FUNCTION ASSEMBLE_BYTE_FROM_QUARTERS (* this Function combines the 4 QUARTER BYTES to a BYTE *)
  (* Standard: 61499-1; Description: Copyright (c) 2024 HR Agrartechnik GmbH This program and the accompanying materials are made available under the terms of the Eclipse Public License 2.0 which is available at https://www.eclipse.org/legal/epl-2.0/ SPDX-License-Identifier: EPL-2.0 *)
  (* Version 3.0, 2025-04-14, Patrick Aigner, changed package *)
  (* Version 1.1, 2024-07-28, Moritz Ortmeier, HR Agrartechnik, rename Function and change Input/Output Variables *)
  (* Version 1.0, 2024-02-22, Franz H??pfinger, HR Agrartechnik, initial Implementation *)
  PACKAGE eclipse4diac::utils::assembling;
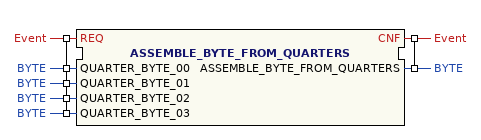
  EVENT_INPUT
    REQ WITH QUARTER_BYTE_00, QUARTER_BYTE_01, QUARTER_BYTE_02, QUARTER_BYTE_03;
  END_EVENT
  EVENT_OUTPUT
    CNF WITH ASSEMBLE_BYTE_FROM_QUARTERS;
  END_EVENT
  VAR_INPUT
    QUARTER_BYTE_00 : BYTE;
    QUARTER_BYTE_01 : BYTE;
    QUARTER_BYTE_02 : BYTE;
    QUARTER_BYTE_03 : BYTE;
  END_VAR
  VAR_OUTPUT
    ASSEMBLE_BYTE_FROM_QUARTERS : BYTE;
  END_VAR
  BODY IN ST:
(* this Function combines the 4 QUARTER BYTES to a BYTE *)
FUNCTION ASSEMBLE_BYTE_FROM_QUARTERS : BYTE

VAR_INPUT
	QUARTER_BYTE_00 : BYTE;
	QUARTER_BYTE_01 : BYTE;
	QUARTER_BYTE_02 : BYTE;
	QUARTER_BYTE_03 : BYTE;
END_VAR

ASSEMBLE_BYTE_FROM_QUARTERS := quarterconst::BYTE_QUARTER_ZZ;
ASSEMBLE_BYTE_FROM_QUARTERS := ASSEMBLE_BYTE_FROM_QUARTERS OR SHL(QUARTER_BYTE_03, quarterconst::SHIFT_QUARTER_03);
ASSEMBLE_BYTE_FROM_QUARTERS := ASSEMBLE_BYTE_FROM_QUARTERS OR SHL(QUARTER_BYTE_02, quarterconst::SHIFT_QUARTER_02);
ASSEMBLE_BYTE_FROM_QUARTERS := ASSEMBLE_BYTE_FROM_QUARTERS OR SHL(QUARTER_BYTE_01, quarterconst::SHIFT_QUARTER_01);
ASSEMBLE_BYTE_FROM_QUARTERS := ASSEMBLE_BYTE_FROM_QUARTERS OR SHL(QUARTER_BYTE_00, quarterconst::SHIFT_QUARTER_00);

END_FUNCTION
  END_BODY
END_FUNCTION
